SUBAPPLICATION Uebung_070 (* WBSD auf UT ausgeben *)
  (* Standard: 61499-2 *)
  (* Version 1.0, 2023-10-23, franz *)
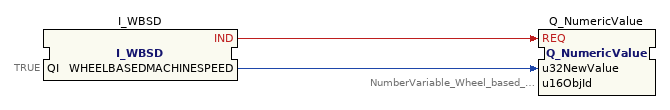
  FBS
    I_WBSD : I_WBSD(QI := TRUE);
    Q_NumericValue : Q_NumericValue(u16ObjId := NumberVariable_Wheel_based_machine_speed);
  END_FBS
  EVENT_CONNECTIONS
    I_WBSD.IND TO Q_NumericValue.REQ;
  END_CONNECTIONS
  DATA_CONNECTIONS
    I_WBSD.WHEELBASEDMACHINESPEED TO Q_NumericValue.u32NewValue;
  END_CONNECTIONS
END_SUBAPPLICATION
